(* CoDeSys 2.3.9.50 project: 2B.pr6 *)
(* Libraries: STANDARD.LB6 5.6.98 12:03:02 *)

(* POU MAIN, LD *)
PROGRAM MAIN
VAR
	H AT %QX0.0: BOOL;
	A AT %IX0.0: BOOL;
	E AT %IX0.4: BOOL;
	F AT %IX0.5: BOOL;
	G AT %IX0.6: BOOL;
	C AT %IX0.2: BOOL;
	D AT %IX0.3: BOOL;
END_VAR
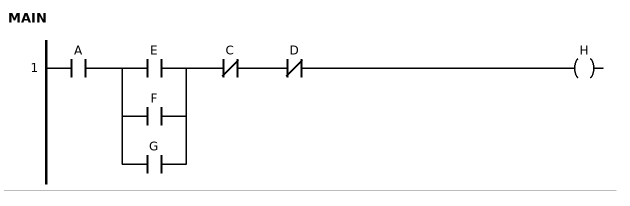
_LD_ (* Ladder Diagram *)
NETWORK 1
	[A] - { [E] | [F] | [G] } - [/C] - [/D] --- (H)
_END_LD_
(* the same logic as Structured Text *)
(* Network 1 *)
H := A AND (E OR F OR G) AND NOT C AND NOT D;
END_PROGRAM

(* Visualisation Q2B
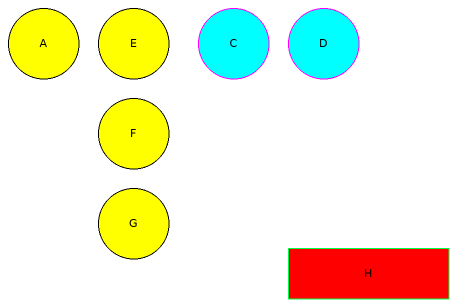
ellipse at (30,100)-(101,171): text "A"; alarm colour if %IX0.0; toggles %IX0.0
ellipse at (120,100)-(191,171): text "E"; alarm colour if %IX0.4; toggles %IX0.4
ellipse at (120,190)-(191,261): text "F"; alarm colour if %IX0.5; toggles %IX0.5
ellipse at (220,100)-(291,171): text "C"; alarm colour if %IX0.2; toggles %IX0.2
ellipse at (310,100)-(381,171): text "D"; alarm colour if %IX0.3; toggles %IX0.3
ellipse at (120,280)-(191,351): text "G"; alarm colour if %IX0.6; toggles %IX0.6
rectangle at (310,340)-(471,391): text "H"; alarm colour if %QX0.0; toggles %QX0.0
*)
